// TIA Portal V19 export
DATA_BLOCK "DB_Parameters"   // DB2
{ S7_Optimized_Access := 'TRUE'; DB_Accessible_From_OPC_UA := 'FALSE' }
// stored: DBAccessibleFromOPCUA false, DBAccessibleFromWebserver false, MemoryReserve 100
   VAR RETAIN
      SensorParameter42B4 { ExternalAccessible := 'False'; ExternalVisible := 'False'; ExternalWritable := 'False'} : "stConfigScaleIntReal";   // Parameter for sensor car body detection (42B4 & 42B3)
      SwitchSensorValue { ExternalAccessible := 'False'; ExternalVisible := 'False'; ExternalWritable := 'False'} : Real := 650.0;   // Level parameter switch for car body detection
      uiSpeedLockEccentric { ExternalAccessible := 'False'; ExternalVisible := 'False'; ExternalWritable := 'False'} : UInt := 50;   // Rotation speed for lock eccentric
      RemoveSandPaperParam { ExternalAccessible := 'False'; ExternalVisible := 'False'; ExternalWritable := 'False'} : "stFerRoboticParam";   // FerRobotic parameter for remove the wor sandpaper
      PickUpSandPaperParam { ExternalAccessible := 'False'; ExternalVisible := 'False'; ExternalWritable := 'False'} : "stFerRoboticParam";   // FerRobotic parameter for pich up a new sandpaper
      FlatnessCtrlParam { ExternalAccessible := 'False'; ExternalVisible := 'False'; ExternalWritable := 'False'} : "stFerRoboticParam";   // FerRobotic paramter for flatness contrl disk planeity
      ConfigGreaseZaxis { ExternalAccessible := 'False'; ExternalVisible := 'False'; ExternalWritable := 'False'} : "stConfigGrease";
      ConfigGreaseXaxis { ExternalAccessible := 'False'; ExternalVisible := 'False'; ExternalWritable := 'False'} : "stConfigGrease";
      ConfigVacuumValve { ExternalAccessible := 'False'; ExternalVisible := 'False'; ExternalWritable := 'False'} : "stConfigActuator";
      tTimeoutGimball { ExternalAccessible := 'False'; ExternalVisible := 'False'; ExternalWritable := 'False'} : Time := T#5S;
      tTimeoutEccentric { ExternalAccessible := 'False'; ExternalVisible := 'False'; ExternalWritable := 'False'} : Time := T#20S;
      rFlatnessStrockPos { ExternalAccessible := 'False'; ExternalVisible := 'False'; ExternalWritable := 'False'} : Real := 23.9;   // FerRobotic strock position for control flatness
      rDeltaFlatnessStrock { ExternalAccessible := 'False'; ExternalVisible := 'False'; ExternalWritable := 'False'} : Real := 0.8;   // Delta maxi for flatness control
      nNbDiskLeft { ExternalAccessible := 'False'; ExternalVisible := 'False'; ExternalWritable := 'False'} : USInt := 1;
      nNbDiskRight { ExternalAccessible := 'False'; ExternalVisible := 'False'; ExternalWritable := 'False'} : USInt := 2;
      rLowLimiteStroke { ExternalAccessible := 'False'; ExternalVisible := 'False'; ExternalWritable := 'False'} : Real := 5.0;
      StrokeTooExtend { ExternalAccessible := 'False'; ExternalVisible := 'False'; ExternalWritable := 'False'} : "stHysteresis";
      StrokeTooRetract { ExternalAccessible := 'False'; ExternalVisible := 'False'; ExternalWritable := 'False'} : "stHysteresis";
   END_VAR
BEGIN
   SensorParameter42B4.nInputMin := 0;
   SensorParameter42B4.nIntputMax := 27648;
   SensorParameter42B4.xUniPolar := TRUE;
   SensorParameter42B4.xReverseValue := TRUE;
   SensorParameter42B4.rOutputMin := 200.0;
   SensorParameter42B4.rOutputMax := 1000.0;
   SensorParameter42B4.rOffsetFixe := 0.0;
   SensorParameter42B4.rOffsetProp := 1.0;
   RemoveSandPaperParam.nSetForceTarget := 20;
   RemoveSandPaperParam.nSetForceZero := 10;
   RemoveSandPaperParam.usiSetTimeRamp := 0;
   RemoveSandPaperParam.uiSetSpeed := 0;
   PickUpSandPaperParam.nSetForceTarget := 100;
   PickUpSandPaperParam.nSetForceZero := 0;
   PickUpSandPaperParam.usiSetTimeRamp := 0;
   PickUpSandPaperParam.uiSetSpeed := 0;
   FlatnessCtrlParam.nSetForceTarget := 20;
   FlatnessCtrlParam.nSetForceZero := 0;
   FlatnessCtrlParam.usiSetTimeRamp := 0;
   FlatnessCtrlParam.uiSetSpeed := 0;
   ConfigGreaseZaxis.uiNbPulsePerKm := 4411;
   ConfigGreaseZaxis.uiKmForGreasing := 32;
   ConfigGreaseZaxis.tTimeEnableGreasePump := T#1M;
   ConfigGreaseZaxis.tTimeoutPxGrease := T#1M;
   ConfigGreaseXaxis.uiNbPulsePerKm := 4411;
   ConfigGreaseXaxis.uiKmForGreasing := 32;
   ConfigGreaseXaxis.tTimeEnableGreasePump := T#2M;
   ConfigGreaseXaxis.tTimeoutPxGrease := T#2M;
   ConfigVacuumValve.xEnaMeasureTimeHome := FALSE;
   ConfigVacuumValve.xEnaMeasureTimeAction := FALSE;
   ConfigVacuumValve.xKeepHomeSolActive := FALSE;
   ConfigVacuumValve.xKeepActionSolActive := TRUE;
   ConfigVacuumValve.xPresHomePxSensor := TRUE;
   ConfigVacuumValve.xPresActionPxSensor := TRUE;
   ConfigVacuumValve.tSwitchingCommand := T#50MS;
   ConfigVacuumValve.tTimeOutHomeSensor := T#8S;
   ConfigVacuumValve.tTimeOutActionSensor := T#8S;
   ConfigVacuumValve.tHomeTime := T#3S;
   ConfigVacuumValve.tActionTime := T#3S;
   ConfigVacuumValve.tFilterPxHome := T#100MS;
   ConfigVacuumValve.tFilterPxAction := T#100MS;
   StrokeTooExtend.rValueOn := 40.0;
   StrokeTooExtend.rValueOff := 35.0;
   StrokeTooRetract.rValueOn := 8.0;
   StrokeTooRetract.rValueOff := 13.0;
END_DATA_BLOCK
